Staubli VAL3: loadPath.pgx

program loadPath(bool& x_bRes, string x_sFile)
begin
  //加载路径
  x_bRes=false
  if prd:libLoad(sFolder+x_sFile)!=0
    logMsg(sItem+":加载失败")
    popUpMsg(sItem+":加载失败")
    return
  endIf
  x_bRes=true

end
